// TIA Portal V21 export
// export: Created 2026-07-11T14:49:10.285131Z, ExportSetting None, DisplayName Totally Integrated Automation Portal, DisplayVersion V21, DisplayName SINAMICS Startdrive Advanced, DisplayVersion V21, DisplayName SINAMICS Startdrive G110M, G120, G120C, G120D, G120P, G115D, DisplayVersion V21, DisplayName SINAMICS Startdrive G130, G150, S120, S150, G200, G220, S200, S210, S220, Innomotics MVD, DisplayVersion V21, DisplayName STEP 7 Professional, DisplayVersion V21, DisplayName STEP 7 Safety, DisplayVersion V21, DisplayName Tech WebApplication, DisplayVersion V21, DisplayName WinCC Basic/Comfort/Advanced, DisplayVersion V21, DisplayName WinCC Professional, DisplayVersion V21, DisplayName WinCC Unified, DisplayVersion V21
FUNCTION_BLOCK "MotionControl_LAD"   // FB2102, LAD
{ S7_Optimized_Access := 'TRUE' }
// stored: AutoNumber false, MemoryReserve 100, SetENOAutomatically false
   VAR_INPUT
      Exe_MC_Reset : Bool;
      En_MC_Power : Bool;
      Exe_MC_Home : Bool;
      Exe_JogFwd : Bool;
      Exe_JogBwd : Bool;
      Exe_MC_Abs : Bool;
      Exe_Halt : Bool;
      Sp_MC_Home_Position : Real;
      Sp_MC_Home_Mode : Int;
      Sp_MC_Power_StartMode : Int := 1;
      Sp_MC_Power_StopMode : Int;
      Sp_MC_Jog_Velocity : Real := 10.0;
      Sp_MC_Abs_Position : Real;
      Sp_MC_Abs_Velocity : Real := 10.0;
   END_VAR
   VAR_OUTPUT
      Output_ActVelocity : Real;
      Output_ActPosition : Real;
      Output_StandStill : Bool;
      Output_MC_Error : Bool;
      Output_MC_Power_Status : Bool;
      Output_MC_Abs_Done : Bool;
      Output_MC_Abs_Busy : Bool;
   END_VAR
   VAR_IN_OUT
      AxisTO : TO_PositioningAxis;
   END_VAR
   VAR
      AxisReady_PosAxis : Bool;
      MC_Reset_Instance { S7_SetPoint := 'True'} : MC_Reset;
      MC_Home_Instance { S7_SetPoint := 'True'} : MC_Home;
      MC_Power_Instance { S7_SetPoint := 'True'} : MC_Power;
      MC_MoveJog_Instance { S7_SetPoint := 'True'} : MC_MoveJog;
      MC_Halt_Instance { S7_SetPoint := 'True'} : MC_Halt;
      MC_MoveAbsolute_Instance { S7_SetPoint := 'True'} : MC_MoveAbsolute;
   END_VAR
   VAR CONSTANT
      ADAPTED : DInt := 2;
      NOT_APPLICABLE : DInt := 3;
   END_VAR
BEGIN

REGION Network 1: MC_Reset
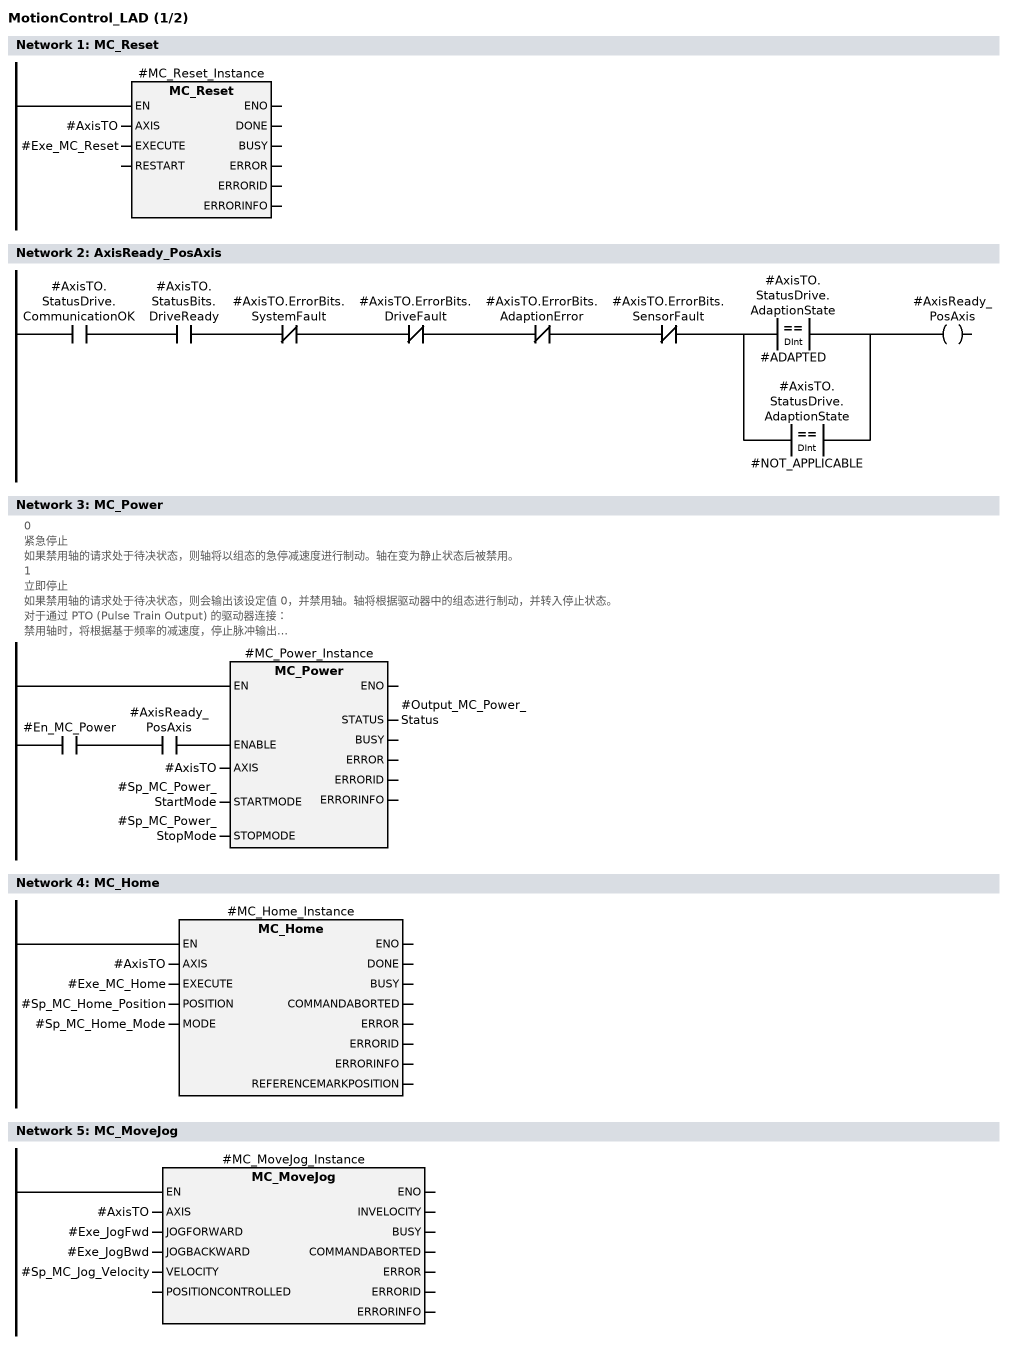
   RUNG wire#powerrail
      #MC_Reset_Instance.MC_Reset(Axis := #AxisTO, Execute := #Exe_MC_Reset, Restart :=, Done =>, Busy =>, Error =>, ErrorID =>, ErrorInfo =>)
   END_RUNG
   // the same network as SCL:
   #MC_Reset_Instance(Axis := #AxisTO, Execute := #Exe_MC_Reset);   // MC_Reset
END_REGION

REGION Network 2: AxisReady_PosAxis
   RUNG wire#powerrail
      Contact( #AxisTO.StatusDrive.CommunicationOK )
      Contact( #AxisTO.StatusBits.DriveReady )
      I_Contact( #AxisTO.ErrorBits.SystemFault )
      I_Contact( #AxisTO.ErrorBits.DriveFault )
      I_Contact( #AxisTO.ErrorBits.AdaptionError )
      I_Contact( #AxisTO.ErrorBits.SensorFault )
      wire#w1
      { S7_Templates := "SrcType := DInt" } EQ_Contact(in1 := #AxisTO.StatusDrive.AdaptionState, in2 := #ADAPTED)
      wire#w2
      Coil( #AxisReady_PosAxis )
   END_RUNG
   RUNG wire#w1
      { S7_Templates := "SrcType := DInt" } EQ_Contact(in1 := #AxisTO.StatusDrive.AdaptionState, in2 := #NOT_APPLICABLE)
   END_RUNG wire#w2
   // the same network as SCL:
   #AxisReady_PosAxis := #AxisTO.StatusDrive.CommunicationOK AND #AxisTO.StatusBits.DriveReady AND NOT #AxisTO.ErrorBits.SystemFault AND NOT #AxisTO.ErrorBits.DriveFault AND NOT #AxisTO.ErrorBits.AdaptionError AND NOT #AxisTO.ErrorBits.SensorFault AND ((#AxisTO.StatusDrive.AdaptionState = #ADAPTED) OR (#AxisTO.StatusDrive.AdaptionState = #NOT_APPLICABLE));
END_REGION

REGION Network 3: MC_Power
   // 0
   // 紧急停止
   // 
   // 如果禁用轴的请求处于待决状态，则轴将以组态的急停减速度进行制动。轴在变为静止状态后被禁用。
   // 
   // 1
   // 立即停止
   // 
   // 如果禁用轴的请求处于待决状态，则会输出该设定值 0，并禁用轴。轴将根据驱动器中的组态进行制动，并转入停止状态。
   // 
   // 对于通过 PTO (Pulse Train Output) 的驱动器连接：
   // 禁用轴时，将根据基于频率的减速度，停止脉冲输出：
   // 
   // 输出频率 ≥ 100 Hz
   // 
   // 减速度：最长 30 ms
   // 
   // 输出频率 < 100 Hz
   // 
   // 减速度：30 ms；2 Hz 时，最长 1.5 s
   // 
   // 2
   // 
   // 带有加速度变化率控制的紧急停止
   // 
   // 如果禁用轴的请求处于待决状态，则轴将以组态的急停减速度进行制动。如果激活了加速度变化率控制，会将已组态的加速度变化率考虑在内。轴在变为静止状态后被禁用。
   RUNG wire#powerrail
      #MC_Power_Instance.MC_Power(Enable := wire#w1, Axis := #AxisTO, StartMode := #Sp_MC_Power_StartMode, StopMode := #Sp_MC_Power_StopMode, Status => #Output_MC_Power_Status, Busy =>, Error =>, ErrorID =>, ErrorInfo =>)
   END_RUNG
   RUNG wire#powerrail
      Contact( #En_MC_Power )
      Contact( #AxisReady_PosAxis )
   END_RUNG wire#w1
   // the same network as SCL:
   #MC_Power_Instance(Enable := #En_MC_Power AND #AxisReady_PosAxis,   // MC_Power
                      Axis := #AxisTO,
                      StartMode := #Sp_MC_Power_StartMode,
                      StopMode := #Sp_MC_Power_StopMode,
                      Status => #Output_MC_Power_Status);
END_REGION

REGION Network 4: MC_Home
   RUNG wire#powerrail
      #MC_Home_Instance.MC_Home(Axis := #AxisTO, Execute := #Exe_MC_Home, Position := #Sp_MC_Home_Position, Mode := #Sp_MC_Home_Mode, Done =>, Busy =>, CommandAborted =>, Error =>, ErrorID =>, ErrorInfo =>, ReferenceMarkPosition =>)
   END_RUNG
   // the same network as SCL:
   #MC_Home_Instance(Axis := #AxisTO,   // MC_Home
                     Execute := #Exe_MC_Home,
                     Position := #Sp_MC_Home_Position,
                     Mode := #Sp_MC_Home_Mode);
END_REGION

REGION Network 5: MC_MoveJog
   RUNG wire#powerrail
      #MC_MoveJog_Instance.MC_MoveJog(Axis := #AxisTO, JogForward := #Exe_JogFwd, JogBackward := #Exe_JogBwd, Velocity := #Sp_MC_Jog_Velocity, PositionControlled :=, InVelocity =>, Busy =>, CommandAborted =>, Error =>, ErrorID =>, ErrorInfo =>)
   END_RUNG
   // the same network as SCL:
   #MC_MoveJog_Instance(Axis := #AxisTO,   // MC_MoveJog
                        JogForward := #Exe_JogFwd,
                        JogBackward := #Exe_JogBwd,
                        Velocity := #Sp_MC_Jog_Velocity);
END_REGION

REGION Network 6: MC_MoveAbsolute
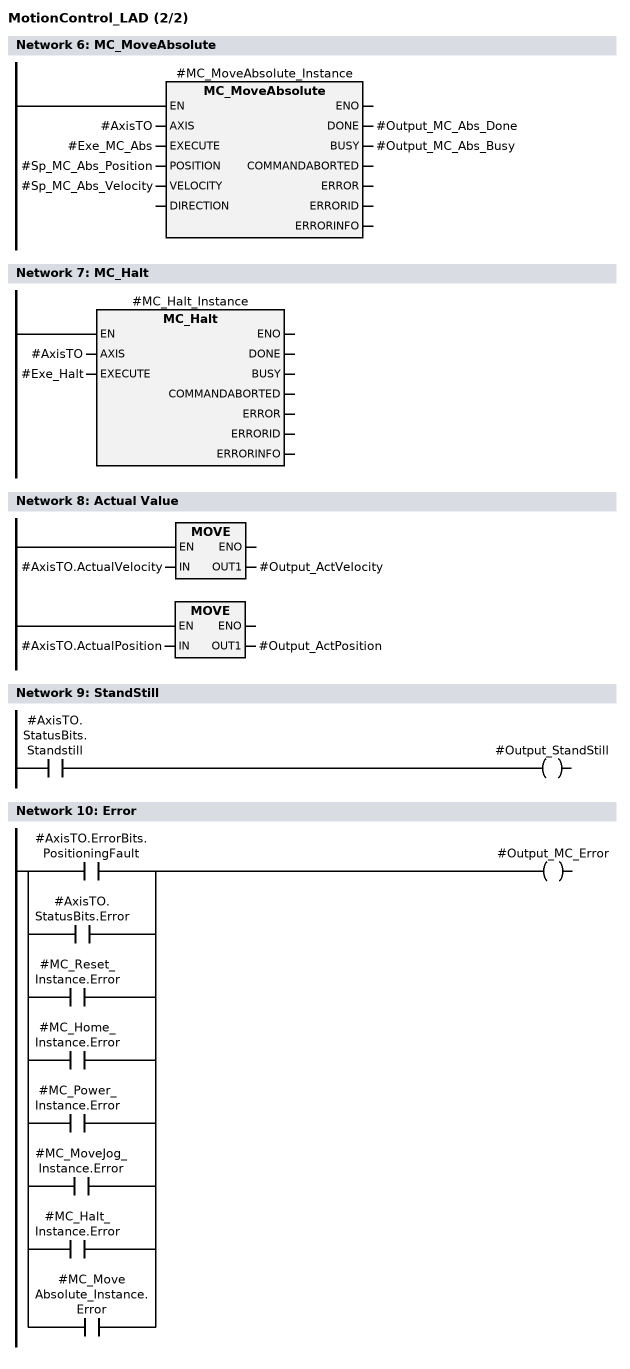
   RUNG wire#powerrail
      #MC_MoveAbsolute_Instance.MC_MoveAbsolute(Axis := #AxisTO, Execute := #Exe_MC_Abs, Position := #Sp_MC_Abs_Position, Velocity := #Sp_MC_Abs_Velocity, Direction :=, Done => #Output_MC_Abs_Done, Busy => #Output_MC_Abs_Busy, CommandAborted =>, Error =>, ErrorID =>, ErrorInfo =>)
   END_RUNG
   // the same network as SCL:
   #MC_MoveAbsolute_Instance(Axis := #AxisTO,   // MC_MoveAbsolute
                           Execute := #Exe_MC_Abs,
                           Position := #Sp_MC_Abs_Position,
                           Velocity := #Sp_MC_Abs_Velocity,
                           Done => #Output_MC_Abs_Done,
                           Busy => #Output_MC_Abs_Busy);
END_REGION

REGION Network 7: MC_Halt
   RUNG wire#powerrail
      #MC_Halt_Instance.MC_Halt(Axis := #AxisTO, Execute := #Exe_Halt, Done =>, Busy =>, CommandAborted =>, Error =>, ErrorID =>, ErrorInfo =>)
   END_RUNG
   // the same network as SCL:
   #MC_Halt_Instance(Axis := #AxisTO, Execute := #Exe_Halt);   // MC_Halt
END_REGION

REGION Network 8: Actual Value
   RUNG wire#powerrail
      Move(in := #AxisTO.ActualVelocity, out1 => #Output_ActVelocity)
   END_RUNG
   RUNG wire#powerrail
      Move(in := #AxisTO.ActualPosition, out1 => #Output_ActPosition)
   END_RUNG
   // the same network as SCL:
   #Output_ActVelocity := #AxisTO.ActualVelocity;
   #Output_ActPosition := #AxisTO.ActualPosition;
END_REGION

REGION Network 9: StandStill
   RUNG wire#powerrail
      Contact( #AxisTO.StatusBits.Standstill )
      Coil( #Output_StandStill )
   END_RUNG
   // the same network as SCL:
   #Output_StandStill := #AxisTO.StatusBits.Standstill;
END_REGION

REGION Network 10: Error
   RUNG wire#powerrail
      Contact( #AxisTO.ErrorBits.PositioningFault )
      wire#w1
      Coil( #Output_MC_Error )
   END_RUNG
   RUNG wire#powerrail
      Contact( #AxisTO.StatusBits.Error )
   END_RUNG wire#w1
   RUNG wire#powerrail
      Contact( #MC_Reset_Instance.Error )
   END_RUNG wire#w1
   RUNG wire#powerrail
      Contact( #MC_Home_Instance.Error )
   END_RUNG wire#w1
   RUNG wire#powerrail
      Contact( #MC_Power_Instance.Error )
   END_RUNG wire#w1
   RUNG wire#powerrail
      Contact( #MC_MoveJog_Instance.Error )
   END_RUNG wire#w1
   RUNG wire#powerrail
      Contact( #MC_Halt_Instance.Error )
   END_RUNG wire#w1
   RUNG wire#powerrail
      Contact( #MC_MoveAbsolute_Instance.Error )
   END_RUNG wire#w1
   // the same network as SCL:
   #Output_MC_Error := #AxisTO.ErrorBits.PositioningFault OR #AxisTO.StatusBits.Error OR #MC_Reset_Instance.Error OR #MC_Home_Instance.Error OR #MC_Power_Instance.Error OR #MC_MoveJog_Instance.Error OR #MC_Halt_Instance.Error OR #MC_MoveAbsolute_Instance.Error;
END_REGION
END_FUNCTION_BLOCK
